(* CoDeSys 2.3.9.412 project: test.pro *)
(* Libraries: STANDARD.LIB 4.10.05 11:14:46, IECSFC.LIB 13.4.06 15:51:28, ANALYZATION.LIB 5.10.99 09:05:06 *)

(* PLC configuration (modules and I/O channels)
Fast discrete inputs [I_SIMPLE_INPUT] node 0, in %IB0 out %QB0 {Filtrationtime = 10; Visibility = No}
  AT %IX0.0 [BitInput] Discrete input 1
  AT %IX0.1 [BitInput] Discrete input 2
Discrete inputs - 16 [ID130] node 1, in %IB1 out %QB1 {Filtrationtime_GeneralINP = 10; Visibility = No; PinCount = 16}
  AT %IB1.0 [ByteInput] 8 discrete inputs
  AT %IB1.1 [ByteInput] 8 discrete inputs
Fast discrete outputs [OWEN_ID570] node 2, in %IB2 out %QB2 {SafeValueBool = FALSE; SafeValueBool = FALSE; SafeValueBool = FALSE; SafeValueBool = FALSE; Visibility = No}
  OUT1 AT %QX2.0 [BitOutput] Fast discrete output 1
  OUT2 AT %QX2.1 [BitOutput] Fast discrete output 2
  OUT3 AT %QX2.2 [BitOutput] Fast discrete output 3
  AT %QX2.3 [BitOutput] Fast discrete output 4
Discrete outputs - 8 [ID131] node 3, in %IB3 out %QB3 {SafeValueByte = 0; Visibility = No; PinCount = 10}
  AT %QB3.0 [ByteOutput] 8 discrete outputs
Special input [ID103] node 4, in %IB4 out %QB4 {Filtrationtime = 1000; PinCount = 1; WatchDogPeriod = 400; PollPeriod = 3000; Visibility = No}
  AT %IX4.0 [BitInput] Special input
Special output [ID104] node 5, in %IB5 out %QB5 {Visibility = No; PinCount = 1}
  AT %QX5.0 [BitOutput] Special output
*)

(* POU PLC_PRG, CFC *)
PROGRAM PLC_PRG
VAR
	IN4: BOOL;
	gate: BOOL;
	leak: BOOL;
	emergency: BOOL;
END_VAR
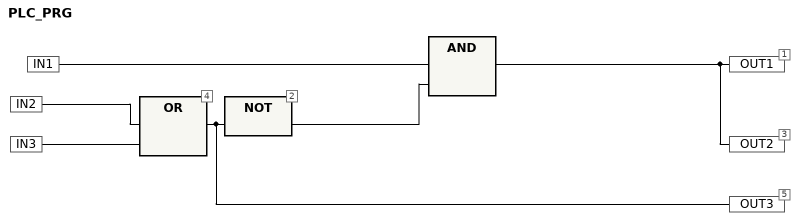
_CFC_ (* Continuous Function Chart, elements in execution order *)
#0 AND(IN1, #2)
#1 OUT1 <= #0
#2 NOT(#4)
#3 OUT2 <= #0
#4 OR(IN2, IN3)
#5 OUT3 <= #4
_END_CFC_
END_PROGRAM

(* Visualisation main
1 more shapes without text or variables
1 elements of other kinds (tables, trends, ...) not read
*)
